// TIA Portal V20 export
DATA_BLOCK "F-DB_Laser"   // DB140, F_DB
// stored: AutoNumber false, InstanceOfName F-FB_Laser, InstanceOfType FB
"F-FB_Laser"
   // VAR
   //    FDBACK_LaserPowerSupply : FDBACK;
   //    FDBACK_Shutter : FDBACK;
   //    sFeedBackShutter : Bool;
   //    sAckFdbShutter : Bool;
   //    sLaserSupplyPower : Bool;
   //    sAckFdbPowLaser : Bool;
   //    sPositiveFrontButtonShutter : Bool;
   //    sNegativeFrontMaintenanceDoor : Bool;
   //    sNegativeFrontDoor : Bool;
   //    sNegativeRoofLeftDoor : Bool;
   //    sNegativeRoofRightDoor : Bool;
   //    sNegativeLaserExternDoor : Bool;
   //    sNegativeSasOneDoor : Bool;
   // END_VAR
BEGIN
END_DATA_BLOCK
